{attribute 'OPC.UA.DA' := '1'}
{attribute 'OPC.UA.DA.StructuredType' := '1'}
{attribute 'OPC.UA.AdditionalStructuredType.NamespaceName' := 'http://beckhoff.com/UA/TE6100_OpcUa_NodesetEditor_Sample_Types/'}
{attribute 'OPC.UA.AdditionalStructuredType.Id' := 's=<StructuredDataType>:ST_Complex_2'}
{attribute 'pack_mode' := '1'}
TYPE ST_Complex_2 :
STRUCT
	c1 		: ST_Complex_1;
	s_5 	: STRING[5]; (*String, max 5 chars*)
	e 		: E_Enum_1;
	s_3 	: STRING[3]; (*String, max 3 chars*)
	cArr 	: ARRAY[0..5] OF ST_Complex_1;
	iArr 	: ARRAY[0..100] OF DINT;	
END_STRUCT
END_TYPE

(* stored: Version 1.1.0.1
   DUT ST_Complex_2: Id {e3a263a3-b266-46c7-bf3b-e050c8a2f76f} *)
